FUNCTION_BLOCK FB_SendEmail
VAR_INPUT
	sAlarmName: STRING(255);
	bStart: BOOL;
END_VAR
VAR_OUTPUT
	bNTProcessBusy:BOOL;
END_VAR
VAR
	NT_StartProcess: NT_StartProcess;
	sPath: STRING := 'C:\DAT\ExecutableFiles\Sendemail.bat ';
	sPath2: STRING := 'C:\DAT\ExecutableFiles';
	bNTErr: BOOL;

	dummy: BOOL;
END_VAR

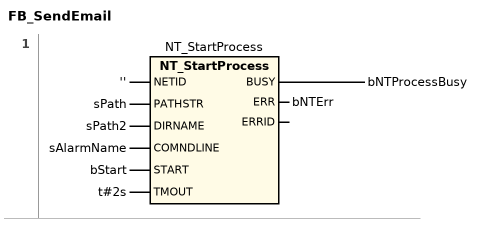
// NETWORK 1
NT_StartProcess(
    NETID := '',
    PATHSTR := sPath,
    DIRNAME := sPath2,
    COMNDLINE := sAlarmName,
    START := bStart,
    TMOUT := t#2s,
    ERR => bNTErr);
bNTProcessBusy := NT_StartProcess.BUSY;

END_FUNCTION_BLOCK

(* stored: Version 1.1.0.1, ProductVersion 3.1.4024.9
   POU FB_SendEmail: Id {d1734b2f-b923-4bfe-80f0-f8f6b878ab17}, SpecialFunc None *)
